// TIA Portal V17 export
// export: Created 2025-06-26T06:49:28.5348487Z, ExportSetting WithDefaults, DisplayName Totally Integrated Automation Portal, DisplayVersion V17 Update 8, DisplayName TIA Portal Openness, DisplayVersion V17 Update 8, DisplayName TIA Portal Version Control Interface, DisplayVersion V17, DisplayName STEP 7 Professional, DisplayVersion V17 Update 8, DisplayName STEP 7 Safety, DisplayVersion V17 Update 6, DisplayName WinCC Advanced, DisplayVersion V17 Update 8
TYPE "stET200AL_RTD"
// stored: IsFailsafeCompliant false
   STRUCT
      CH00 : Int;
      CH01 : Int;
      CH02 : Int;
      CH03 : Int;
      CH00_ok : Bool;
      CH01_ok : Bool;
      CH02_ok : Bool;
      CH03_ok : Bool;
   END_STRUCT;
END_TYPE
